# EPICS substitutions: utcaApp/Db/rtmlamp.substitutions
file db/scan_task.template {
    {}
}

file db/rtmlamp.template {
    pattern {RTM_CHAN ADDR}
    {"M1:PS-FCH", "0"}
    {"M1:PS-FCV", "1"}
    {"M2:PS-FCH", "2"}
    {"M2:PS-FCV", "3"}
    {"C2:PS-FCH", "4"}
    {"C2:PS-FCV", "5"}
    {"C3:PS-FCH", "6"}
    {"C3:PS-FCV", "7"}
    {"XX:PS-FC0", "8"}
    {"XX:PS-FC0", "9"}
    {"XX:PS-FC1", "10"}
    {"XX:PS-FC1", "11"}
}
